Fanuc KAREL source: kt00136.KL

-- PROVISIONAL review KL for V1013-1; original PC SHA256 3edfb5f4927b091774239fcfec50ed8c7ceed9c41cc5e029909d979afaf6f22d
-- Incomplete behavior may be omitted. Consult companion uncertainty JSON. Do not deploy.
PROGRAM KT00136
%NOLOCKGROUP
VAR
  I1 : INTEGER
  OUT : REAL
-- UNRESOLVED_DECL H2 type=002017
BEGIN
  -- UNRESOLVED_PC offsets 5-16; opcodes 2E,23
  -- UNRESOLVED_PC offsets 21-35; opcodes 2E,22,9D,33,B4
  -- UNRESOLVED_PC offsets 40-63; opcodes 21,22,9D,33,B3,55,64,23
  -- UNRESOLVED_PC offsets 68-72; opcodes 7F
END KT00136
